{attribute 'GeneratedUsingTerminal: EL3773-0000-0021'}
{attribute addProperty BoxType "EL3773-0000-0021"}
{attribute addProperty Id "I3_SamplesAT %I*I3_Samples_2549228720"}
{attribute addProperty CRC "3110368094"}
{attribute addProperty Size "20"}
TYPE L3_Current_Samples_B964735E EXTENDS TcoIo.InputBase_8311D824 :
STRUCT
	{attribute addProperty Name "I3_Samples"}
	I3_Samples AT %I* : I3_Samples_25492287;
END_STRUCT
END_TYPE

(* stored: Version 1.2.0.0, ProductVersion 3.1.4024.11
   DUT L3_Current_Samples_B964735E: Id {9b3b663a-7cdd-0b57-1c4a-9ef57e9ac0ae} *)
